(*	Extending the base block

*)
FUNCTION_BLOCK OopExmplExtension EXTENDS OopExmplBase
VAR_INPUT
	I_Extension:BOOL;
END_VAR
VAR_OUTPUT
	Q_Extension:BOOL;
END_VAR
VAR
	HM_Extension:BOOL;
END_VAR

//call baseblock functionality
SUPER^();

//extra code added by extension
HM_Extension := HM_Base AND I_Extension;
Q_Extension := HM_Extension;

END_FUNCTION_BLOCK

(* stored: Version 1.1.0.1
   POU OopExmplExtension: Id {007eade0-4d94-0c6a-11e2-9da8f294431c}, SpecialFunc None *)
